TYPE ST_NovramData :
STRUCT
END_STRUCT
END_TYPE

(* stored: Version 1.1.0.1, ProductVersion 3.1.4020.12
   DUT ST_NovramData: Id {f84d6aa2-8eb8-42b2-ad96-ebeb99948569} *)
